(* PLC project  *)

CONFIGURATION FSOE_2
END_CONFIGURATION
